// TIA Portal V21 export
FUNCTION_BLOCK "FB309"   // FB309, LAD
TITLE = FB309
{ S7_Optimized_Access := 'FALSE' }
AUTHOR : PRECISE
FAMILY : PRECISE
// RAW MATERIAL ADDITION LIQUID DRUM
// stored: AutoNumber false, SetENOAutomatically false
   VAR_INPUT
      Enable : Bool;
      Disable : Bool;
      Fault : Bool;
      SecPulse : Bool;
      AlwaysTrue : Bool;
      StartConfirmationPopupSel : Bool;   // StartConfirmationPopupSel: 0-NO/1-YES
      EndConfirmationPopupSel : Bool;   // EndConfirmationPopupSel: 0-NO/1-YES
      WeightBasedSel : Bool;   // Weight Based Sel: 0-NO/1-YES
      AdditionMethodSel : Bool;   // Addition Method : 0-Add In Weight/1-Loss In Weight
      RMAddPopupSel : Bool;   // RM Add Popup Sel: 0-NO/1-YES
      SetQuantity : Real := 10.0;   // Weight Based Sel: 1-YES
      SetSpeed : Real := 50.0;
      ActualQuantity : Real;   // Collecting Vessel Weight
      ActualQuantityRMVessel : Real;   // Transffering Vessel Weight
      InflightQuantity : Real;
      DelaytoStartPump : Int := 3;
   END_VAR
   VAR_OUTPUT
      LineValves : Bool;
      PumpCmd : Bool;
      StartConfirmationPopup : Bool;   // For Start Confirmation Popup Selection: Yes
      EndConfirmationPopup : Bool;   // For End Confirmation Popup Selection: Yes
      RMAddPopup : Bool;   // For RMAddPopupSel: 1-YES
      ActualSpeed : Real;
      PrintTrigger : Bool;
      PrintWord : Int;
      PrintStatus : String[50];
   END_VAR
   VAR_IN_OUT
      Start : Bool;
      Stop : Bool;
      Reset : Bool;
      StartConfirmationAck : Bool;   // For Start Confirmation Popup Selection: Yes
      EndConfirmationAck : Bool;   // For End Confirmation Popup Selection: Yes
      RMAddAck : Bool;   // For RMAddPopupSel: 1-YES
      SpareBtn1 : Bool;
      SpareBtn2 : Bool;
      Running : Bool;
      Selected : Bool;
      Paused : Bool;
      StartConfirmationPopupTemp : Bool;   // For Start Confirmation Popup Selection: Yes
      EndConfirmationPopupTemp : Bool;   // For End Confirmation Popup Selection: Yes
      RMAddPopupTemp : Bool;   // For RMAddPopupSel: 1-YES
      RMAddStarted : Bool;
      RMAddOver : Bool;
      ActualSetQuantityCalc : Real;   // For WeightBaseSel: 1-YES
      ActualSetQuantity : Real;   // For WeightBaseSel: 1-YES
   END_VAR
   VAR
      ValveOnDelayPV : Int;
      ValveOffDelayPV : Int;
      PrintTriggerTemp : Bool;
      RE1 : Bool;
      RE2 : Bool;
      RE3 : Bool;
      RE4 : Bool;
      RE5 : Bool;
      RE6 : Bool;
      RE7 : Bool;
      RE8 : Bool;
      PrintTriggerResetTimer { S7_SetPoint := 'True'} : TON_TIME;
      BtnResetTimer { S7_SetPoint := 'True'} : TON_TIME;
      NameRM : String[40];
   END_VAR
   VAR_TEMP
      STATUS1 : String[40];
      STATUS2 : String[40];
      STATUS3 : String[40];
      STATUS4 : String[40];
      STATUS5 : String[40];
   END_VAR
   VAR_TEMP   // added for the SCL form of the ladder/FBD networks
      _w1 : Bool;
      _w2 : Bool;
      _w3 : Bool;
      _w4 : Bool;
      _w5 : Bool;
      _w6 : Bool;
      _w7 : Bool;
   END_VAR
BEGIN

REGION Network 1: Running
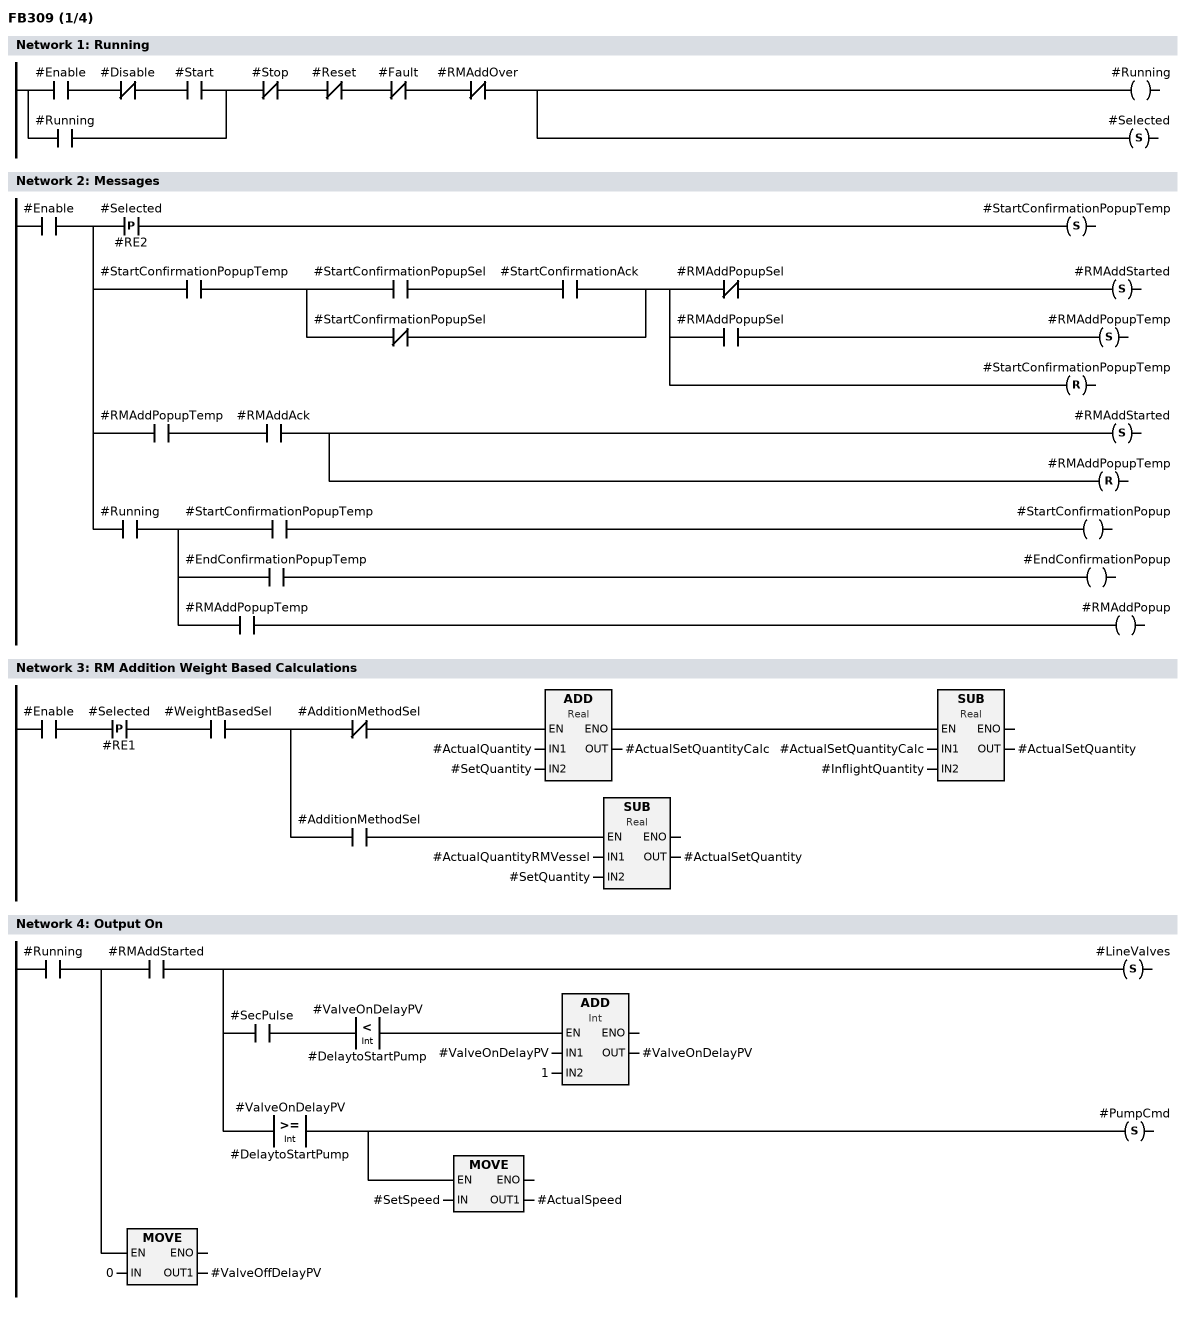
   RUNG wire#powerrail
      Contact( #Enable )
      I_Contact( #Disable )
      Contact( #Start )
      wire#w1
      I_Contact( #Stop )
      I_Contact( #Reset )
      I_Contact( #Fault )
      I_Contact( #RMAddOver )
      wire#w2
      Coil( #Running )
   END_RUNG
   RUNG wire#powerrail
      Contact( #Running )
   END_RUNG wire#w1
   RUNG wire#w2
      S_Coil( #Selected )
   END_RUNG
   // the same network as SCL:
   #Running := ((#Enable AND NOT #Disable AND #Start) OR #Running) AND NOT #Stop AND NOT #Reset AND NOT #Fault AND NOT #RMAddOver;
   IF #Running THEN #Selected := TRUE; END_IF;
END_REGION

REGION Network 2: Messages
   RUNG wire#powerrail
      Contact( #Enable )
      wire#w1
      P_Contact(operand := #Selected, bit := #RE2)
      S_Coil( #StartConfirmationPopupTemp )
   END_RUNG
   RUNG wire#w1
      Contact( #StartConfirmationPopupTemp )
      wire#w2
      Contact( #StartConfirmationPopupSel )
      Contact( #StartConfirmationAck )
      wire#w3
      I_Contact( #RMAddPopupSel )
      S_Coil( #RMAddStarted )
   END_RUNG
   RUNG wire#w2
      I_Contact( #StartConfirmationPopupSel )
   END_RUNG wire#w3
   RUNG wire#w3
      Contact( #RMAddPopupSel )
      S_Coil( #RMAddPopupTemp )
   END_RUNG
   RUNG wire#w3
      R_Coil( #StartConfirmationPopupTemp )
   END_RUNG
   RUNG wire#w1
      Contact( #RMAddPopupTemp )
      Contact( #RMAddAck )
      wire#w4
      S_Coil( #RMAddStarted )
   END_RUNG
   RUNG wire#w4
      R_Coil( #RMAddPopupTemp )
   END_RUNG
   RUNG wire#w1
      Contact( #Running )
      wire#w5
      Contact( #StartConfirmationPopupTemp )
      Coil( #StartConfirmationPopup )
   END_RUNG
   RUNG wire#w5
      Contact( #EndConfirmationPopupTemp )
      Coil( #EndConfirmationPopup )
   END_RUNG
   RUNG wire#w5
      Contact( #RMAddPopupTemp )
      Coil( #RMAddPopup )
   END_RUNG
   // the same network as SCL:
   #_w1 := #Enable AND #Selected AND NOT #RE2;   // rising edge of #Selected
   #RE2 := #Selected;
   IF #_w1 THEN #StartConfirmationPopupTemp := TRUE; END_IF;
   #_w2 := #Enable AND #StartConfirmationPopupTemp AND ((#StartConfirmationPopupSel AND #StartConfirmationAck) OR NOT #StartConfirmationPopupSel);
   IF #_w2 AND NOT #RMAddPopupSel THEN #RMAddStarted := TRUE; END_IF;
   IF #_w2 AND #RMAddPopupSel THEN #RMAddPopupTemp := TRUE; END_IF;
   IF #_w2 THEN #StartConfirmationPopupTemp := FALSE; END_IF;
   IF #Enable AND #RMAddPopupTemp AND #RMAddAck THEN
       #RMAddStarted := TRUE;
       #RMAddPopupTemp := FALSE;
   END_IF;
   #_w3 := #Enable AND #Running;
   #StartConfirmationPopup := #_w3 AND #StartConfirmationPopupTemp;
   #EndConfirmationPopup := #_w3 AND #EndConfirmationPopupTemp;
   #RMAddPopup := #_w3 AND #RMAddPopupTemp;
END_REGION

REGION Network 3: RM Addition Weight Based Calculations
   RUNG wire#powerrail
      Contact( #Enable )
      P_Contact(operand := #Selected, bit := #RE1)
      Contact( #WeightBasedSel )
      wire#w1
      I_Contact( #AdditionMethodSel )
      { S7_Templates := "SrcType := Real"; S7_GenerateENO := "TRUE" } Add(in1 := #ActualQuantity, in2 := #SetQuantity, out => #ActualSetQuantityCalc)
      { S7_Templates := "SrcType := Real"; S7_GenerateENO := "TRUE" } Sub(in1 := #ActualSetQuantityCalc, in2 := #InflightQuantity, out => #ActualSetQuantity)
   END_RUNG
   RUNG wire#w1
      Contact( #AdditionMethodSel )
      { S7_Templates := "SrcType := Real"; S7_GenerateENO := "TRUE" } Sub(in1 := #ActualQuantityRMVessel, in2 := #SetQuantity, out => #ActualSetQuantity)
   END_RUNG
   // the same network as SCL:
   // ENO of a box is taken as its EN; it also drops when the box reports an error
   #_w1 := #Enable AND #Selected AND NOT #RE1;   // rising edge of #Selected
   #RE1 := #Selected;
   #_w2 := #_w1 AND #WeightBasedSel;
   IF #_w2 AND NOT #AdditionMethodSel THEN
       #ActualSetQuantityCalc := #ActualQuantity + #SetQuantity;
       #ActualSetQuantity := #ActualSetQuantityCalc - #InflightQuantity;
   END_IF;
   IF #_w2 AND #AdditionMethodSel THEN #ActualSetQuantity := #ActualQuantityRMVessel - #SetQuantity; END_IF;
END_REGION

REGION Network 4: Output On
   RUNG wire#powerrail
      Contact( #Running )
      wire#w1
      Contact( #RMAddStarted )
      wire#w2
      S_Coil( #LineValves )
   END_RUNG
   RUNG wire#w2
      Contact( #SecPulse )
      { S7_Templates := "SrcType := Int" } LT_Contact(in1 := #ValveOnDelayPV, in2 := #DelaytoStartPump)
      { S7_Templates := "SrcType := Int"; S7_GenerateENO := "TRUE" } Add(in1 := #ValveOnDelayPV, in2 := 1, out => #ValveOnDelayPV)
   END_RUNG
   RUNG wire#w2
      { S7_Templates := "SrcType := Int" } GE_Contact(in1 := #ValveOnDelayPV, in2 := #DelaytoStartPump)
      wire#w3
      S_Coil( #PumpCmd )
   END_RUNG
   RUNG wire#w3
      Move(in := #SetSpeed, out1 => #ActualSpeed)
   END_RUNG
   RUNG wire#w1
      { S7_GenerateENO := "TRUE" } Move(in := 0, out1 => #ValveOffDelayPV)
   END_RUNG
   // the same network as SCL:
   #_w1 := #Running AND #RMAddStarted;
   IF #_w1 THEN #LineValves := TRUE; END_IF;
   IF #_w1 AND #SecPulse AND (#ValveOnDelayPV < #DelaytoStartPump) THEN
       #ValveOnDelayPV := #ValveOnDelayPV + 1;
   END_IF;
   IF #_w1 AND (#ValveOnDelayPV >= #DelaytoStartPump) THEN
       #PumpCmd := TRUE;
       #ActualSpeed := #SetSpeed;
   END_IF;
   IF #Running THEN #ValveOffDelayPV := 0; END_IF;
END_REGION

REGION Network 5: Output Off
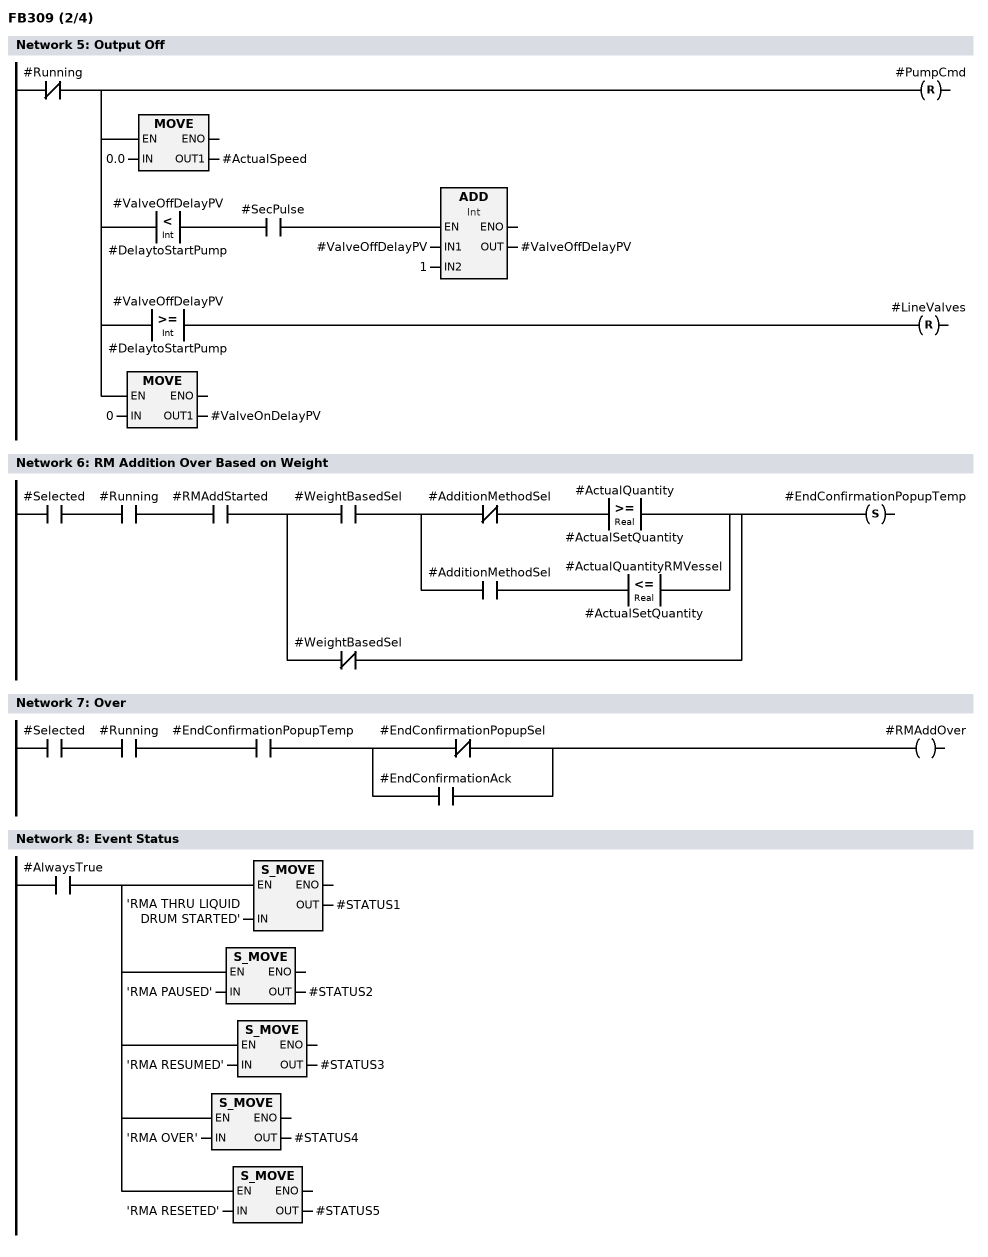
   RUNG wire#powerrail
      I_Contact( #Running )
      wire#w1
      R_Coil( #PumpCmd )
   END_RUNG
   RUNG wire#w1
      Move(in := 0.0, out1 => #ActualSpeed)
   END_RUNG
   RUNG wire#w1
      { S7_Templates := "SrcType := Int" } LT_Contact(in1 := #ValveOffDelayPV, in2 := #DelaytoStartPump)
      Contact( #SecPulse )
      { S7_Templates := "SrcType := Int"; S7_GenerateENO := "TRUE" } Add(in1 := #ValveOffDelayPV, in2 := 1, out => #ValveOffDelayPV)
   END_RUNG
   RUNG wire#w1
      { S7_Templates := "SrcType := Int" } GE_Contact(in1 := #ValveOffDelayPV, in2 := #DelaytoStartPump)
      R_Coil( #LineValves )
   END_RUNG
   RUNG wire#w1
      { S7_GenerateENO := "TRUE" } Move(in := 0, out1 => #ValveOnDelayPV)
   END_RUNG
   // the same network as SCL:
   IF NOT #Running THEN
       #PumpCmd := FALSE;
       #ActualSpeed := 0.0;
   END_IF;
   IF NOT #Running AND (#ValveOffDelayPV < #DelaytoStartPump) AND #SecPulse THEN
       #ValveOffDelayPV := #ValveOffDelayPV + 1;
   END_IF;
   IF NOT #Running AND (#ValveOffDelayPV >= #DelaytoStartPump) THEN #LineValves := FALSE; END_IF;
   IF NOT #Running THEN #ValveOnDelayPV := 0; END_IF;
END_REGION

REGION Network 6: RM Addition Over Based on Weight
   RUNG wire#powerrail
      Contact( #Selected )
      Contact( #Running )
      Contact( #RMAddStarted )
      wire#w1
      Contact( #WeightBasedSel )
      wire#w2
      I_Contact( #AdditionMethodSel )
      { S7_Templates := "SrcType := Real" } GE_Contact(in1 := #ActualQuantity, in2 := #ActualSetQuantity)
      wire#w3
      S_Coil( #EndConfirmationPopupTemp )
   END_RUNG
   RUNG wire#w2
      Contact( #AdditionMethodSel )
      { S7_Templates := "SrcType := Real" } LE_Contact(in1 := #ActualQuantityRMVessel, in2 := #ActualSetQuantity)
   END_RUNG wire#w3
   RUNG wire#w1
      I_Contact( #WeightBasedSel )
   END_RUNG wire#w3
   // the same network as SCL:
   IF #Selected AND #Running AND #RMAddStarted AND ((#WeightBasedSel AND ((NOT #AdditionMethodSel AND (#ActualQuantity >= #ActualSetQuantity)) OR (#AdditionMethodSel AND (#ActualQuantityRMVessel <= #ActualSetQuantity)))) OR NOT #WeightBasedSel) THEN
       #EndConfirmationPopupTemp := TRUE;
   END_IF;
END_REGION

REGION Network 7: Over
   RUNG wire#powerrail
      Contact( #Selected )
      Contact( #Running )
      Contact( #EndConfirmationPopupTemp )
      wire#w1
      I_Contact( #EndConfirmationPopupSel )
      wire#w2
      Coil( #RMAddOver )
   END_RUNG
   RUNG wire#w1
      Contact( #EndConfirmationAck )
   END_RUNG wire#w2
   // the same network as SCL:
   #RMAddOver := #Selected AND #Running AND #EndConfirmationPopupTemp AND (NOT #EndConfirmationPopupSel OR #EndConfirmationAck);
END_REGION

REGION Network 8: Event Status
   RUNG wire#powerrail
      Contact( #AlwaysTrue )
      wire#w1
      S_Move(in := 'RMA THRU LIQUID DRUM STARTED', out => #STATUS1)
   END_RUNG
   RUNG wire#w1
      S_Move(in := 'RMA PAUSED', out => #STATUS2)
   END_RUNG
   RUNG wire#w1
      S_Move(in := 'RMA RESUMED', out => #STATUS3)
   END_RUNG
   RUNG wire#w1
      S_Move(in := 'RMA OVER', out => #STATUS4)
   END_RUNG
   RUNG wire#w1
      S_Move(in := 'RMA RESETED', out => #STATUS5)
   END_RUNG
   // the same network as SCL:
   IF #AlwaysTrue THEN
       #STATUS1 := 'RMA THRU LIQUID DRUM STARTED';
       #STATUS2 := 'RMA PAUSED';
       #STATUS3 := 'RMA RESUMED';
       #STATUS4 := 'RMA OVER';
       #STATUS5 := 'RMA RESETED';
   END_IF;
END_REGION

REGION Network 9: Print Logic
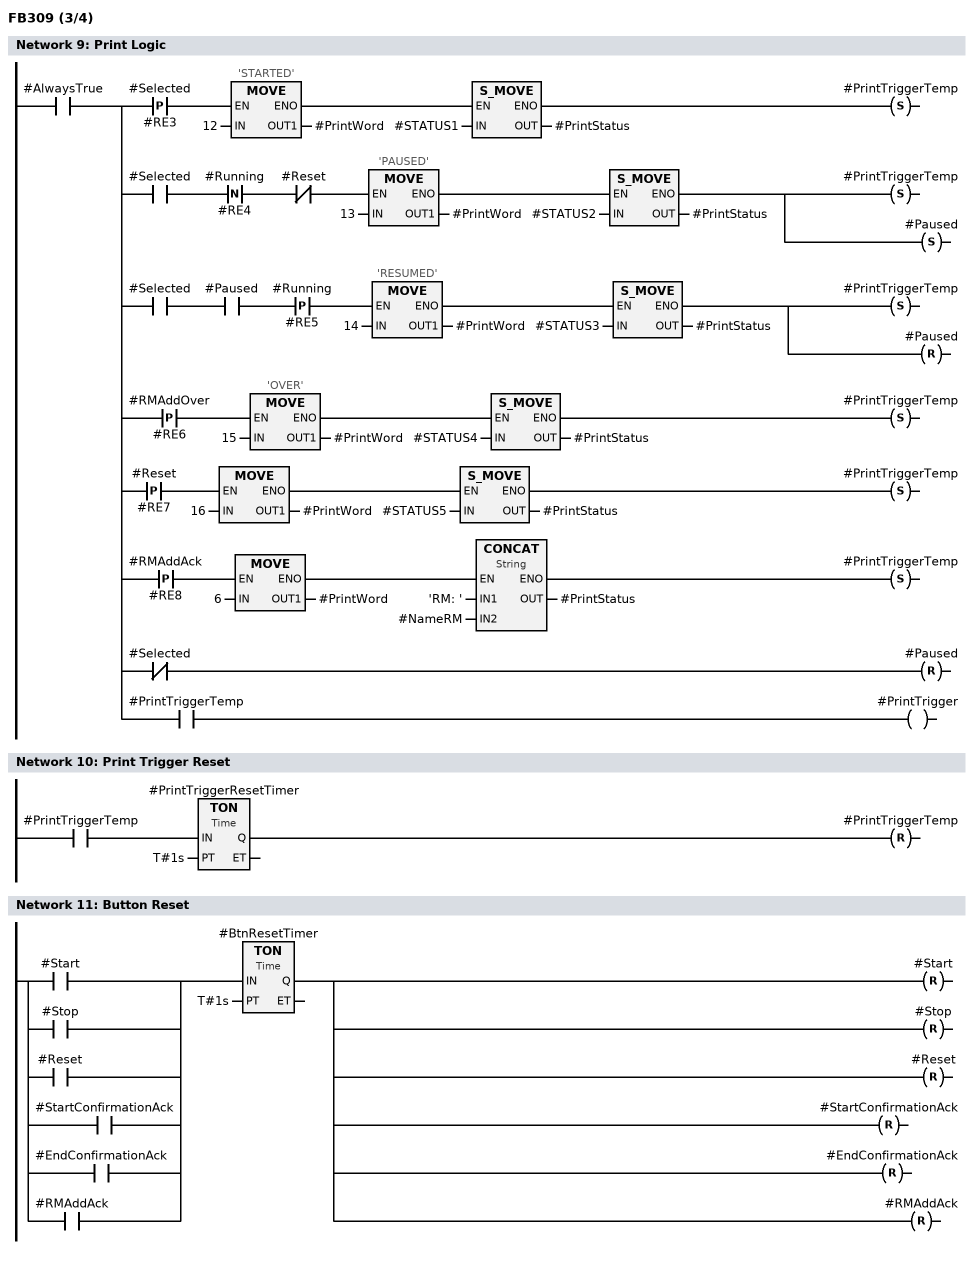
   RUNG wire#powerrail
      Contact( #AlwaysTrue )
      wire#w1
      P_Contact(operand := #Selected, bit := #RE3)
      { S7_GenerateENO := "TRUE" } Move(in := 12, out1 => #PrintWord)   // 'STARTED'
      S_Move(in := #STATUS1, out => #PrintStatus)
      S_Coil( #PrintTriggerTemp )
   END_RUNG
   RUNG wire#w1
      Contact( #Selected )
      N_Contact(operand := #Running, bit := #RE4)
      I_Contact( #Reset )
      { S7_GenerateENO := "TRUE" } Move(in := 13, out1 => #PrintWord)   // 'PAUSED'
      S_Move(in := #STATUS2, out => #PrintStatus)
      wire#w2
      S_Coil( #PrintTriggerTemp )
   END_RUNG
   RUNG wire#w2
      S_Coil( #Paused )
   END_RUNG
   RUNG wire#w1
      Contact( #Selected )
      Contact( #Paused )
      P_Contact(operand := #Running, bit := #RE5)
      { S7_GenerateENO := "TRUE" } Move(in := 14, out1 => #PrintWord)   // 'RESUMED'
      S_Move(in := #STATUS3, out => #PrintStatus)
      wire#w3
      S_Coil( #PrintTriggerTemp )
   END_RUNG
   RUNG wire#w3
      R_Coil( #Paused )
   END_RUNG
   RUNG wire#w1
      P_Contact(operand := #RMAddOver, bit := #RE6)
      { S7_GenerateENO := "TRUE" } Move(in := 15, out1 => #PrintWord)   // 'OVER'
      S_Move(in := #STATUS4, out => #PrintStatus)
      S_Coil( #PrintTriggerTemp )
   END_RUNG
   RUNG wire#w1
      P_Contact(operand := #Reset, bit := #RE7)
      { S7_GenerateENO := "TRUE" } Move(in := 16, out1 => #PrintWord)
      S_Move(in := #STATUS5, out => #PrintStatus)
      S_Coil( #PrintTriggerTemp )
   END_RUNG
   RUNG wire#w1
      P_Contact(operand := #RMAddAck, bit := #RE8)
      { S7_GenerateENO := "TRUE" } Move(in := 6, out1 => #PrintWord)
      { S7_Templates := "[card := 2, str_type := String]" } CONCAT(IN1 := 'RM: ', IN2 := #NameRM, OUT => #PrintStatus)
      S_Coil( #PrintTriggerTemp )
   END_RUNG
   RUNG wire#w1
      I_Contact( #Selected )
      R_Coil( #Paused )
   END_RUNG
   RUNG wire#w1
      Contact( #PrintTriggerTemp )
      Coil( #PrintTrigger )
   END_RUNG
   // the same network as SCL:
   // ENO of a box is taken as its EN; it also drops when the box reports an error
   #_w1 := #AlwaysTrue AND #Selected AND NOT #RE3;   // rising edge of #Selected
   #RE3 := #Selected;
   IF #_w1 THEN
       #PrintWord := 12;   // 'STARTED'
       #PrintStatus := #STATUS1;
       #PrintTriggerTemp := TRUE;
   END_IF;
   #_w2 := #AlwaysTrue AND #Selected AND NOT #Running AND #RE4;   // falling edge of #Running
   #RE4 := #Running;
   IF #_w2 AND NOT #Reset THEN
       #PrintWord := 13;   // 'PAUSED'
       #PrintStatus := #STATUS2;
       #PrintTriggerTemp := TRUE;
       #Paused := TRUE;
   END_IF;
   #_w3 := #AlwaysTrue AND #Selected AND #Paused AND #Running AND NOT #RE5;   // rising edge of #Running
   #RE5 := #Running;
   IF #_w3 THEN
       #PrintWord := 14;   // 'RESUMED'
       #PrintStatus := #STATUS3;
       #PrintTriggerTemp := TRUE;
       #Paused := FALSE;
   END_IF;
   #_w4 := #AlwaysTrue AND #RMAddOver AND NOT #RE6;   // rising edge of #RMAddOver
   #RE6 := #RMAddOver;
   IF #_w4 THEN
       #PrintWord := 15;   // 'OVER'
       #PrintStatus := #STATUS4;
       #PrintTriggerTemp := TRUE;
   END_IF;
   #_w5 := #AlwaysTrue AND #Reset AND NOT #RE7;   // rising edge of #Reset
   #RE7 := #Reset;
   IF #_w5 THEN
       #PrintWord := 16;
       #PrintStatus := #STATUS5;
       #PrintTriggerTemp := TRUE;
   END_IF;
   #_w6 := #AlwaysTrue AND #RMAddAck AND NOT #RE8;   // rising edge of #RMAddAck
   #RE8 := #RMAddAck;
   IF #_w6 THEN #PrintWord := 6; END_IF;
   CONCAT(EN := #_w6, IN1 := 'RM: ', IN2 := #NameRM, OUT => #PrintStatus, ENO => #_w7);
   IF #_w7 THEN #PrintTriggerTemp := TRUE; END_IF;
   IF #AlwaysTrue AND NOT #Selected THEN #Paused := FALSE; END_IF;
   #PrintTrigger := #AlwaysTrue AND #PrintTriggerTemp;
END_REGION

REGION Network 10: Print Trigger Reset
   RUNG wire#powerrail
      Contact( #PrintTriggerTemp )
      { S7_Templates := "time_type := Time" } #PrintTriggerResetTimer.TON(pt := T#1s, et =>)
      R_Coil( #PrintTriggerTemp )
   END_RUNG
   // the same network as SCL:
   #PrintTriggerResetTimer(IN := #PrintTriggerTemp, PT := T#1s);   // TON
   IF #PrintTriggerResetTimer.Q THEN #PrintTriggerTemp := FALSE; END_IF;
END_REGION

REGION Network 11: Button Reset
   RUNG wire#powerrail
      Contact( #Start )
      wire#w1
      { S7_Templates := "time_type := Time" } #BtnResetTimer.TON(pt := T#1s, et =>)
      wire#w2
      R_Coil( #Start )
   END_RUNG
   RUNG wire#powerrail
      Contact( #Stop )
   END_RUNG wire#w1
   RUNG wire#powerrail
      Contact( #Reset )
   END_RUNG wire#w1
   RUNG wire#powerrail
      Contact( #StartConfirmationAck )
   END_RUNG wire#w1
   RUNG wire#powerrail
      Contact( #EndConfirmationAck )
   END_RUNG wire#w1
   RUNG wire#powerrail
      Contact( #RMAddAck )
   END_RUNG wire#w1
   RUNG wire#w2
      R_Coil( #Stop )
   END_RUNG
   RUNG wire#w2
      R_Coil( #Reset )
   END_RUNG
   RUNG wire#w2
      R_Coil( #StartConfirmationAck )
   END_RUNG
   RUNG wire#w2
      R_Coil( #EndConfirmationAck )
   END_RUNG
   RUNG wire#w2
      R_Coil( #RMAddAck )
   END_RUNG
   // the same network as SCL:
   #BtnResetTimer(IN := #Start OR #Stop OR #Reset OR #StartConfirmationAck OR #EndConfirmationAck OR #RMAddAck,   // TON
                  PT := T#1s);
   IF #BtnResetTimer.Q THEN
       #Start := FALSE;
       #Stop := FALSE;
       #Reset := FALSE;
       #StartConfirmationAck := FALSE;
       #EndConfirmationAck := FALSE;
       #RMAddAck := FALSE;
   END_IF;
END_REGION

REGION Network 12: Reset
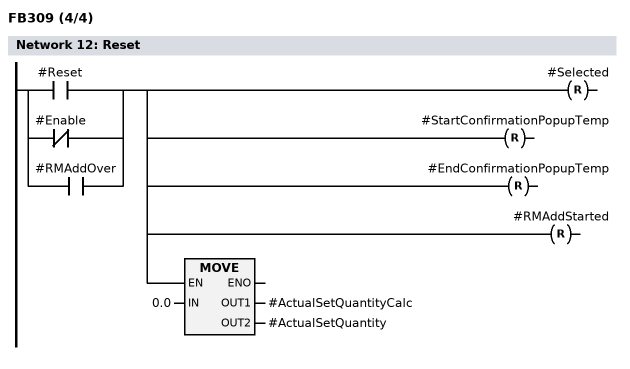
   RUNG wire#powerrail
      Contact( #Reset )
      wire#w1
      R_Coil( #Selected )
   END_RUNG
   RUNG wire#powerrail
      I_Contact( #Enable )
   END_RUNG wire#w1
   RUNG wire#powerrail
      Contact( #RMAddOver )
   END_RUNG wire#w1
   RUNG wire#w1
      R_Coil( #StartConfirmationPopupTemp )
   END_RUNG
   RUNG wire#w1
      R_Coil( #EndConfirmationPopupTemp )
   END_RUNG
   RUNG wire#w1
      R_Coil( #RMAddStarted )
   END_RUNG
   RUNG wire#w1
      Move(in := 0.0, out1 => #ActualSetQuantityCalc, out2 => #ActualSetQuantity)
   END_RUNG
   // the same network as SCL:
   IF #Reset OR NOT #Enable OR #RMAddOver THEN
       #Selected := FALSE;
       #StartConfirmationPopupTemp := FALSE;
       #EndConfirmationPopupTemp := FALSE;
       #RMAddStarted := FALSE;
       #ActualSetQuantityCalc := 0.0;
       #ActualSetQuantity := 0.0;
   END_IF;
END_REGION
END_FUNCTION_BLOCK
